(*********************************** G.D S.p.A. - Technical Department ***********************************
============= PROGRAM INFO ============
FOLDER:             TBD
MACHINES INVOLVED:  TBD 

============= DESCRIPTION =============
csp machine declaration

============= REVISIONS ===============
Date		Version	 	Author      	Description             
----------	-------		------------  	--------------------------------------------
2019/04/05 	0000.00	 	M.Grasso		Creation of the PRG

**********************************************************************************************************)
(*$R process_ref := prc; $*)
PROGRAM csp_case_fc_os_upper
VAR
	
	prc:											process;
	prc_path:										STRING;
	
END_VAR

_read_var_input();

_object_manager();

IF NOT objects_running()
THEN
	RETURN;	
END_IF

_read_process_image();

_mode_manager();

_set_runtime_properties();

(********************************* BODY *********************************)
(************************************************************************)

_handle_messages();

_write_output();

ACTION _handle_messages:
;
END_ACTION

ACTION _handle_process_test:
;
END_ACTION

ACTION _mode_manager:
IF process_mode_req_is_pending(prc)
THEN
    process_apply_mode_req_first_step(prc);
    CASE process_get_mode(prc) OF
        MODE_TO_ABSENT:
			;
        MODE_TO_INACTIVE:
			;
        MODE_TO_TEST:
			;
        MODE_TO_OPERATIONAL:
			;
    END_CASE
    process_apply_mode_req_second_step(prc);
END_IF
END_ACTION

ACTION _object_manager:
IF objects_initialization()
THEN
	sub_process_init(
		object_name					:= 'csp_case_fc_os_upper.prc', 
		process						:= csp_case_flapControl_os.prc, 
		CONVERSION_this				:= prc);
		
	prc_path 						:= process_get_path(prc);
END_IF

IF objects_running()
THEN
	process_cycle(prc);
END_IF
END_ACTION

ACTION _read_process_image:
;
END_ACTION

ACTION _read_var_input:
;
END_ACTION

ACTION _set_runtime_properties:
;
END_ACTION

ACTION _write_output:
;
END_ACTION

END_PROGRAM

(* stored: Version 1.1.0.1, ProductVersion 3.1.4022.12
   POU csp_case_fc_os_upper: Id {4e82e713-2410-4318-aab0-d61737e2f012}, SpecialFunc None
   Action _handle_messages: Id {3a877654-8c4b-40ec-82d1-815c13741d3d}
   Action _handle_process_test: Id {4f09bd00-7e80-4df2-bfd2-5b8a7376b212}
   Action _mode_manager: Id {60b4b4ef-57ee-4b88-9184-6353e1ff9634}
   Action _object_manager: Id {74c073b2-52c6-4f9d-b4af-46b2c0688458}
   Action _read_process_image: Id {a00b6787-a673-4f42-bade-df4b2ee8a617}
   Action _read_var_input: Id {6fc46f27-72bf-42ea-9058-54e41b565cae}
   Action _set_runtime_properties: Id {bc43a989-eb13-460d-872a-11dce3b838da}
   Action _write_output: Id {d98bf18b-0652-40a5-a705-70d645d1abe9} *)
